// TIA Portal V15.1 export
// export: Created 2020-06-12T07:35:42.4287109Z, ExportSetting None, DisplayName Totally Integrated Automation Portal, DisplayVersion V15.1, DisplayName TIA Portal Openness, DisplayVersion V15.1, DisplayName STEP 7 Professional, DisplayVersion V15.1, DisplayName STEP 7 Safety, DisplayVersion V15.1, DisplayName WinCC Advanced, DisplayVersion V15.1
FUNCTION "CW_Common" : Void   // FC1002, FBD
TITLE = CWS [Cooling water system]
{ S7_Optimized_Access := 'TRUE' }
// stored: SetENOAutomatically False
   VAR_TEMP
      tOff : Bool;
      tCWMS1ReqOn : Bool;
      tCWMS2ReqOn : Bool;
      tEconomOff : Bool;
      tNormalCirc : Bool;
   END_VAR
   VAR_TEMP   // added for the SCL form of the ladder/FBD networks
      _w1 : Bool;
   END_VAR
BEGIN

REGION Network 1: MS1 request the pumps
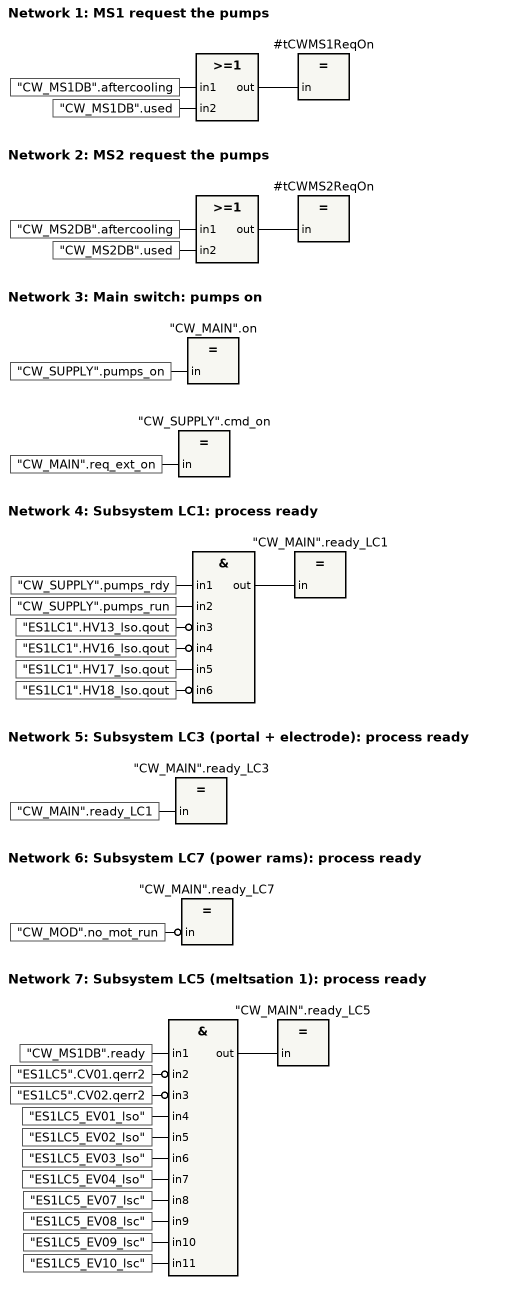
   #tCWMS1ReqOn := "CW_MS1DB".aftercooling OR "CW_MS1DB".used;
END_REGION

REGION Network 2: MS2 request the pumps
   #tCWMS2ReqOn := "CW_MS2DB".aftercooling OR "CW_MS2DB".used;
END_REGION

REGION Network 3: Main switch: pumps on
   "CW_MAIN".on := "CW_SUPPLY".pumps_on;
   "CW_SUPPLY".cmd_on := "CW_MAIN".req_ext_on;
END_REGION

REGION Network 4: Subsystem LC1: process ready
   "CW_MAIN".ready_LC1 := "CW_SUPPLY".pumps_rdy AND "CW_SUPPLY".pumps_run AND NOT "ES1LC1".HV13_lso.qout AND NOT "ES1LC1".HV16_lso.qout AND "ES1LC1".HV17_lso.qout AND NOT "ES1LC1".HV18_lso.qout;
END_REGION

REGION Network 5: Subsystem LC3 (portal + electrode): process ready
   "CW_MAIN".ready_LC3 := "CW_MAIN".ready_LC1;
END_REGION

REGION Network 6: Subsystem LC7 (power rams): process ready
   "CW_MAIN".ready_LC7 := NOT "CW_MOD".no_mot_run;
END_REGION

REGION Network 7: Subsystem LC5 (meltsation 1): process ready
   "CW_MAIN".ready_LC5 := "CW_MS1DB".ready AND NOT "ES1LC5".CV01.qerr2 AND NOT "ES1LC5".CV02.qerr2 AND "ES1LC5_EV01_lso" AND "ES1LC5_EV02_lso" AND "ES1LC5_EV03_lso" AND "ES1LC5_EV04_lso" AND "ES1LC5_EV07_lsc" AND "ES1LC5_EV08_lsc" AND "ES1LC5_EV09_lsc" AND "ES1LC5_EV10_lsc";
END_REGION

REGION Network 8: Subsystem LC6 (meltsation 2): process ready
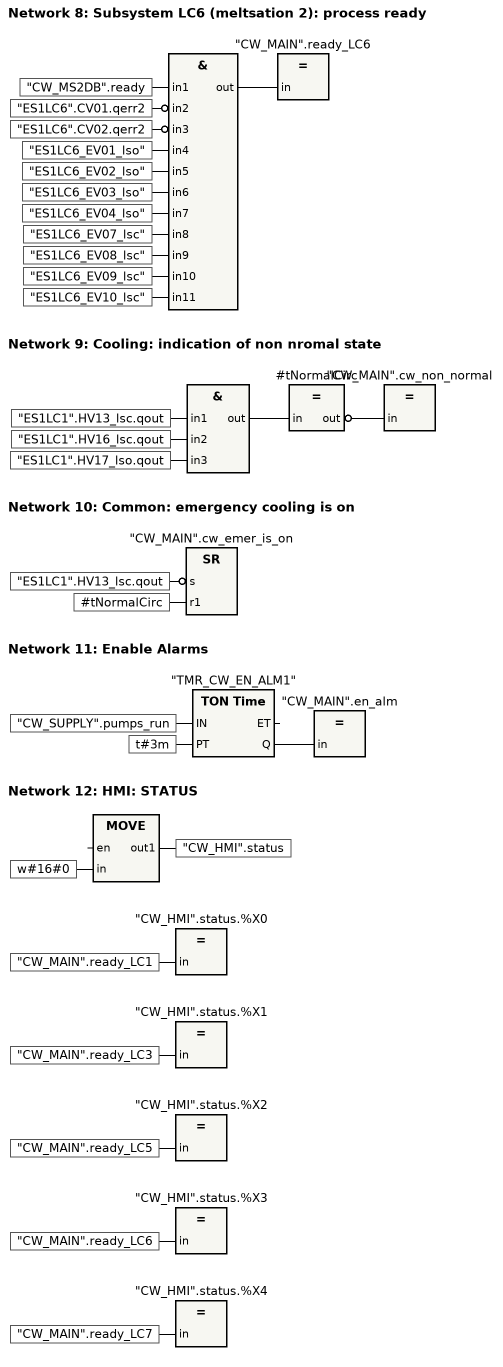
   "CW_MAIN".ready_LC6 := "CW_MS2DB".ready AND NOT "ES1LC6".CV01.qerr2 AND NOT "ES1LC6".CV02.qerr2 AND "ES1LC6_EV01_lso" AND "ES1LC6_EV02_lso" AND "ES1LC6_EV03_lso" AND "ES1LC6_EV04_lso" AND "ES1LC6_EV07_lsc" AND "ES1LC6_EV08_lsc" AND "ES1LC6_EV09_lsc" AND "ES1LC6_EV10_lsc";
END_REGION

REGION Network 9: Cooling: indication of non nromal state
   // This indicator shows a non-normal cooling state: may be a emerencgy cooling was started or may be a after-maintenace error
   #_w1 := "ES1LC1".HV13_lsc.qout AND "ES1LC1".HV16_lsc.qout AND "ES1LC1".HV17_lso.qout;
   #tNormalCirc := #_w1;
   "CW_MAIN".cw_non_normal := NOT #_w1;
END_REGION

REGION Network 10: Common: emergency cooling is on
   IF NOT "ES1LC1".HV13_lsc.qout THEN
       "CW_MAIN".cw_emer_is_on := TRUE;   // SR flip-flop
   END_IF;
   IF #tNormalCirc THEN "CW_MAIN".cw_emer_is_on := FALSE; END_IF;
END_REGION

REGION Network 11: Enable Alarms
   "TMR_CW_EN_ALM1".TON(IN := "CW_SUPPLY".pumps_run, PT := t#3m);
   "CW_MAIN".en_alm := "TMR_CW_EN_ALM1".Q;
END_REGION

REGION Network 12: HMI: STATUS
   "CW_HMI".status := w#16#0;
   "CW_HMI".status.%X0 := "CW_MAIN".ready_LC1;
   "CW_HMI".status.%X1 := "CW_MAIN".ready_LC3;
   "CW_HMI".status.%X2 := "CW_MAIN".ready_LC5;
   "CW_HMI".status.%X3 := "CW_MAIN".ready_LC6;
   "CW_HMI".status.%X4 := "CW_MAIN".ready_LC7;
END_REGION
END_FUNCTION
